Staubli VAL3: start.pgx

public program start()
begin
  // Position des cases
  //   28   29  30  31             ligne 8
  //     ....                      ...
  //  8   9  10  11                ligne 3
  //    4   5   6   7              ligne 2
  //  0   1   2   3                ligne 1
  //pCase[0] = case O en bas à gauche du plateau

  //se met en position 0
  //  call DeplacementInit()

  //Deplacementpion(X,Y) -> deplacement du pion de X vers Y
  //  call Deplacementpion(0,4)

  //call TestPositionCal()

  call DeplacementInit()
  call Data_acqu()

  if TEST[2]==0
    call Deplacementpion(TEST[0],TEST[1])

  else
    call Deplacementpion(TEST[0],TEST[1])
    call Pionperdu(TEST[2],Compteur_perdu)
    Compteur_perdu=Compteur_perdu+1
  endIf
end
